TYPE E_SM_STATUS :
(
	OK		:= 0,
	ERROR
);
END_TYPE

(* stored: Version 1.1.0.1, ProductVersion 3.1.4022.16
   DUT E_SM_STATUS: Id {5dab13c0-db7d-4370-9333-50f9c71f156e} *)
